FUNCTION_BLOCK AX_OR_6 (* FB to calculate boolean OR *)
  (* Standard: 61499-2; Description: Copyright (c) 2024 HR Agrartechnik GmbH This program and the accompanying materials are made available under the terms of the Eclipse Public License 2.0 which is available at https://www.eclipse.org/legal/epl-2.0/ SPDX-License-Identifier: EPL-2.0 *)
  (* Version 1.0, 2024-10-23, Franz Höpfinger, HR Agrartechnik GmbH *)
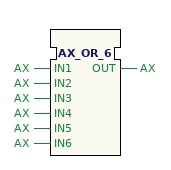
  SOCKETS
    IN1 : AX; (* OR input 1 *)
    IN2 : AX; (* OR input 2 *)
    IN3 : AX; (* OR input 3 *)
    IN4 : AX; (* OR input 4 *)
    IN5 : AX; (* OR input 5 *)
    IN6 : AX; (* OR input 6 *)
  END_SOCKETS
  PLUGS
    OUT : AX; (* OR result *)
  END_PLUGS
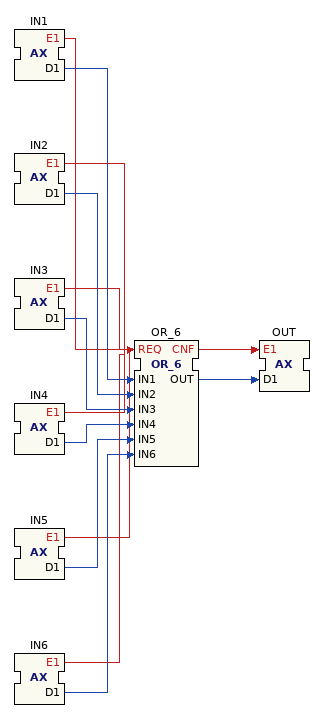
  FBS
    OR_6 : OR_6;
  END_FBS
  EVENT_CONNECTIONS
    IN1.E1 TO OR_6.REQ;
    IN2.E1 TO OR_6.REQ;
    OR_6.CNF TO OUT.E1;
    IN3.E1 TO OR_6.REQ;
    IN4.E1 TO OR_6.REQ;
    IN5.E1 TO OR_6.REQ;
    IN6.E1 TO OR_6.REQ;
  END_CONNECTIONS
  DATA_CONNECTIONS
    IN1.D1 TO OR_6.IN1;
    IN2.D1 TO OR_6.IN2;
    OR_6.OUT TO OUT.D1;
    IN3.D1 TO OR_6.IN3;
    IN4.D1 TO OR_6.IN4;
    IN5.D1 TO OR_6.IN5;
    IN6.D1 TO OR_6.IN6;
  END_CONNECTIONS
END_FUNCTION_BLOCK
